Fanuc KAREL source: KO00032.KL

PROGRAM KO00032
%NOLOCKGROUP
VAR
  P1: JOINTPOS
  P2: JOINTPOS
  P3: JOINTPOS
  P4: JOINTPOS
  OUT: JOINTPOS
BEGIN
  OUT = FRAME(P1, P2, P3, P4)
END KO00032
